// TIA Portal V19 export
VAR_GLOBAL   // PLC tag table "A02_201"
   A0201_Motore_Bancalata_1_Controllo_Connettore AT %I131.3 : Bool;   // 970X1A
   A0201_Banco_1_Phc_Ingresso AT %I131.4 : Bool;   // 973SQ1
   A0201_Banco_1_Phc_Uscita AT %I131.5 : Bool;   // 973SQ2
   "A0201_AUX_Spalla_1.1_Ls_Minimo" AT %I131.6 : Bool;   // 982SQ1
   "A0201_AUX_Spalla_1.1_Ls_Massimo" AT %I131.7 : Bool;   // 982SQ2
   "A0201_AUX_Spalla_1.2_Ls_Minimo" AT %I132.0 : Bool;   // 992SQ1
   "A0201_AUX_Spalla_1.2_Ls_Massimo" AT %I132.1 : Bool;   // 992SQ2
   "A0201_AUX_Spalla_1.3_Ls_Minimo" AT %I132.2 : Bool;   // 1002SQ1
   "A0201_AUX_Spalla_1.3_Ls_Massimo" AT %I132.3 : Bool;   // 1002SQ2
   "A0201_AUX_Spalla_1.4_Ls_Minimo" AT %I132.4 : Bool;   // 1006SQ1
   "A0201_AUX_Spalla_1.4_Ls_Massimo" AT %I132.5 : Bool;   // 1006SQ2
   A0201_Motore_Bancalata_2_Controllo_Connettore AT %I132.6 : Bool;   // 1020X1A
   A0201_Banco_2_Phc_Ingresso AT %I132.7 : Bool;   // 1023SQ1
   A0201_Banco_2_Phc_Uscita AT %I133.0 : Bool;   // 1023SQ2
   "A0201_AUX_Spalla_2.1_Ls_Minimo" AT %I133.1 : Bool;   // 1032SQ1
   "A0201_AUX_Spalla_2.1_Ls_Massimo" AT %I133.2 : Bool;   // 1032SQ2
   "A0201_AUX_Spalla_2.2_Ls_Minimo" AT %I133.3 : Bool;   // 1042SQ1
   "A0201_AUX_Spalla_2.2_Ls_Massimo" AT %I133.4 : Bool;   // 1042SQ2
   A0201_Motore_Bancalata_3_Lato_1_Controllo_Connettore AT %I133.5 : Bool;   // 1060X1A
   A0201_Banco_3_Lato_1_Phc_Ingresso AT %I133.6 : Bool;   // 1063SQ1
   A0201_Banco_3_Lato_1_Phc_Uscita AT %I133.7 : Bool;   // 1063SQ2
   "A0201_AUX_Spalla_3.1_Ls_Minimo_Apertura" AT %I134.0 : Bool;   // 1072SQ1
   "A0201_AUX_Spalla_3.1_Ls_Massimo_Apertura" AT %I134.1 : Bool;   // 1072SQ2
   "A0201_Spalla_3.3_Apre" AT %Q4.4 : Bool;   // 1080KM1
   "A0201_Spalla_3.3_Chiude" AT %Q4.5 : Bool;   // 1080KM2
   "A0201_Spalla_3.3_Anomalia_Termico" AT %I4.1 : Bool;   // 1080QF1
   "A0201_AUX_Spalla_3.3_Ls_Minimo_Apertura" AT %I134.2 : Bool;   // 1081SQ1
   "A0201_AUX_Spalla_3.3_Ls_Massimo_Apertura" AT %I134.3 : Bool;   // 1081SQ2
   "A0201_Spalla_3.5_Apre" AT %Q4.6 : Bool;   // 1085KM1
   "A0201_Spalla_3.5_Chiude" AT %Q4.7 : Bool;   // 1085KM2
   "A0201_Spalla_3.5_Anomalia_Termico" AT %I4.2 : Bool;   // 1085QF1
   "A0201_AUX_Spalla_3.5_Ls_Minimo_Apertura" AT %I134.4 : Bool;   // 1086SQ1
   "A0201_AUX_Spalla_3.5_Ls_Massimo_Apertura" AT %I134.5 : Bool;   // 1086SQ2
   "A0201_Spalla_3.7_Apre" AT %Q5.0 : Bool;   // 1090KM1
   "A0201_Spalla_3.7_Chiude" AT %Q5.1 : Bool;   // 1090KM2
   "A0201_AUX_Spalla_3.7_Ls_Minimo_Apertura" AT %I134.6 : Bool;   // 1091SQ1
   "A0201_AUX_Spalla_3.7_Ls_Massimo_Apertura" AT %I134.7 : Bool;   // 1091SQ2
   A0201_Motore_Bancalata_3_Lato_2_Controllo_Connettore AT %I135.0 : Bool;   // 1110X1A
   A0201_Banco_3_Lato_2_Phc_Ingresso AT %I135.1 : Bool;   // 1113SQ1
   A0201_Banco_3_Lato_2_Phc_Uscita AT %I135.2 : Bool;   // 1113SQ2
   "A0201_AUX_Spalla_3.2_Ls_Minimo" AT %I135.3 : Bool;   // 1122SQ1
   "A0201_AUX_Spalla_3.2_Ls_Massimo" AT %I135.4 : Bool;   // 1122SQ2
   "A0201_Spalla_3.4_Apre" AT %Q5.2 : Bool;   // 1130KM1
   "A0201_Spalla_3.4_Chiude" AT %Q5.3 : Bool;   // 1130KM2
   "A0201_Spalla_3.4_Anomalia_Termico" AT %I4.4 : Bool;   // 1130QF1
   "A0201_AUX_Spalla_3.4_Ls_Minimo" AT %I135.5 : Bool;   // 1131SQ1
   "A0201_AUX_Spalla_3.4_Ls_Massimo" AT %I135.6 : Bool;   // 1131SQ2
   "A0201_Spalla_3.6_Apre" AT %Q5.4 : Bool;   // 1135KM1
   "A0201_Spalla_3.6_Chiude" AT %Q5.5 : Bool;   // 1135KM2
   "A0201_Spalla_3.6_Anomalia_Termico" AT %I4.5 : Bool;   // 1135QF1
   "A0201_AUX_Spalla_3.6_Ls_Minimo" AT %I135.7 : Bool;   // 1136SQ1
   "A0201_AUX_Spalla_3.6_Ls_Massimo" AT %I136.0 : Bool;   // 1136SQ2
   "A0201_Spalla_3.8_Apre" AT %Q5.6 : Bool;   // 1140KM1
   "A0201_Spalla_3.8_Chiude" AT %Q5.7 : Bool;   // 1140KM2
   "A0201_Spalla_3.8_Anomalia_Termico" AT %I4.6 : Bool;   // 1140QF1
   "A0201_AUX_Spalla_3.8_Ls_Minimo" AT %I136.1 : Bool;   // 1141SQ1
   "A0201_AUX_Spalla_3.8_Ls_Massimo" AT %I136.2 : Bool;   // 1141SQ2
   A0201_Ventilatore_Mot_Profila_Marcia AT %Q1.5 : Bool;   // 1192QF1
   A0201_Ventilatore_Mot_Profila_Feedback AT %I4.7 : Bool;   // 1192KM1
   A0201_Phc_Inizio_Indroduttore_Profila AT %I136.3 : Bool;   // 1198SQ1
   A0201_Profila_Controllo_Bancale_Bit0 AT %I136.4 : Bool;   // 1204X1
   A0201_Profila_Controllo_Bancale_Bit1 AT %I136.5 : Bool;   // 1204X1
   A0201_Profila_Controllo_Bancale_Bit2 AT %I136.6 : Bool;   // 1204X1
   A0201_Profila_Phc_Prima_Encoder AT %I136.7 : Bool;   // 1204SQ1
   A0201_Profila_Phc_Dopo_Encoder AT %I137.0 : Bool;   // 1204SQ2
   A0201_Profila_Cassette_Pompa_Lubrificante_Marcia AT %Q1.6 : Bool;   // 1210QF1
   A0201_Profila_Cassette_Pompa_Lubrificante_Feedback AT %I5.0 : Bool;   // 1210KM1
   A0201_Profila_Cassette_V_Sezionatrice_Generale AT %Q140.0 : Bool;   // 1212YV1
   A0201_Profila_Cassette_Livello_Lubrificante AT %I137.1 : Bool;   // 1212SL1
   A0201_Profila_Cassetta_1_V_Lubrificante_1 AT %Q140.1 : Bool;   // 1214YV1
   A0201_Profila_Cassetta_1_V_Lubrificante_2 AT %Q140.2 : Bool;   // 1214YV2
   A0201_Profila_Cassetta_1_V_Lubrificante_3 AT %Q140.3 : Bool;   // 1214YV3
   A0201_Profila_Cassetta_1_V_Feedback_Lubrificante_1 AT %I137.2 : Bool;   // 1214SQ1
   A0201_Profila_Cassetta_1_V_Feedback_Lubrificante_2 AT %I137.3 : Bool;   // 1214SQ2
   A0201_Profila_Cassetta_1_V_Feedback_Lubrificante_3 AT %I137.4 : Bool;   // 1214SQ3
   A0201_Profila_Cassetta_1_V_Lubrificante_4 AT %Q140.4 : Bool;   // 1215YV1
   A0201_Profila_Cassetta_1_V_Lubrificante_5 AT %Q140.5 : Bool;   // 1215YV2
   A0201_Profila_Cassetta_1_V_Lubrificante_6 AT %Q140.6 : Bool;   // 1215YV3
   A0201_Profila_Cassetta_1_V_Feedback_Lubrificante_4 AT %I137.5 : Bool;   // 1215SQ1
   A0201_Profila_Cassetta_1_V_Feedback_Lubrificante_5 AT %I137.6 : Bool;   // 1215SQ2
   A0201_Profila_Cassetta_1_V_Feedback_Lubrificante_6 AT %I137.7 : Bool;   // 1215SQ3
   A0201_Profila_Cassetta_2_V_Lubrificante_1 AT %Q140.7 : Bool;   // 1218YV1
   A0201_Profila_Cassetta_2_V_Lubrificante_2 AT %Q141.0 : Bool;   // 1218YV2
   A0201_Profila_Cassetta_2_V_Lubrificante_3 AT %Q141.1 : Bool;   // 1218YV3
   A0201_Profila_Cassetta_2_V_Feedback_Lubrificante_1 AT %I138.0 : Bool;   // 1218SQ1
   A0201_Profila_Cassetta_2_V_Feedback_Lubrificante_2 AT %I138.1 : Bool;   // 1218SQ2
   A0201_Profila_Cassetta_2_V_Feedback_Lubrificante_3 AT %I138.2 : Bool;   // 1218SQ3
   A0201_Profila_Cassetta_2_V_Lubrificante_4 AT %Q141.2 : Bool;   // 1219YV1
   A0201_Profila_Cassetta_2_V_Lubrificante_5 AT %Q141.3 : Bool;   // 1219YV2
   A0201_Profila_Cassetta_2_V_Lubrificante_6 AT %Q141.4 : Bool;   // 1219YV3
   A0201_Profila_Cassetta_2_V_Feedback_Lubrificante_4 AT %I138.3 : Bool;   // 1219SQ1
   A0201_Profila_Cassetta_2_V_Feedback_Lubrificante_5_Libero AT %I138.4 : Bool;   // 1219SQ2
   A0201_Profila_Cassetta_2_V_Feedback_Lubrificante_6_Libero AT %I138.5 : Bool;   // 1219SQ3
   A0201_Profila_Cassetta_3_V_Lubrificante_1 AT %Q141.5 : Bool;   // 1222YV1
   A0201_Profila_Cassetta_3_V_Lubrificante_2 AT %Q141.6 : Bool;   // 1222YV2
   A0201_Profila_Cassetta_3_V_Lubrificante_3 AT %Q141.7 : Bool;   // 1222YV3
   A0201_Profila_Cassetta_3_V_Feedback_Lubrificante_1 AT %I138.6 : Bool;   // 1222SQ1
   A0201_Profila_Cassetta_3_V_Feedback_Lubrificante_2 AT %I138.7 : Bool;   // 1222SQ2
   A0201_Profila_Cassetta_3_V_Feedback_Lubrificante_3 AT %I139.0 : Bool;   // 1222SQ3
   A0201_Profila_Cassetta_3_V_Lubrificante_4 AT %Q142.0 : Bool;   // 1223YV1
   A0201_Profila_Cassetta_3_V_Lubrificante_5 AT %Q142.1 : Bool;   // 1223YV2
   A0201_Profila_Cassetta_3_V_Lubrificante_6 AT %Q142.2 : Bool;   // 1223YV3
   A0201_Profila_Cassetta_3_V_Feedback_Lubrificante_4 AT %I139.1 : Bool;   // 1223SQ1
   A0201_Profila_Cassetta_3_V_Feedback_Lubrificante_5_Libero AT %I139.2 : Bool;   // 1223SQ2
   A0201_Profila_Cassetta_3_V_Feedback_Lubrificante_6_Libero AT %I139.3 : Bool;   // 1223SQ3
   A0201_Fine_Profila_V_Soffio AT %Q142.3 : Bool;   // 1234YV1
   A0201_Fine_Profila_V_Soffio_Pulizia_Phc_Tacca AT %Q142.4 : Bool;   // 1234YV2
   A0201_Ls_Controllo_Inceppamento AT %I139.4 : Bool;   // 1243SQ1
   A0201_Carrello_Riposizionatore_Phc_Prima_Encoder AT %I139.5 : Bool;   // 1245SQ1
   A0201_Carrello_Misuratore_Posizione_Zero AT %I139.6 : Bool;   // 1245SQ2
   A0201_Carrello_Misuratore_Rallentamento_Verso_Zero AT %I139.7 : Bool;   // 1245SQ3
   A0201_Carrello_Misuratore_Rallentamento_Verso_Posizione_Rest AT %I140.0 : Bool;   // 1245SQ4
   A0201_Carrello_Misuratore_Stop_Verso_Rest AT %I140.1 : Bool;   // 1245SQ5
   A0201_Carrello_Misuratore_Posizione_Work AT %I140.2 : Bool;   // 1245SQ6
   A0201_Carrello_Misuratore_In_Appoggio_Tra_Loro AT %I140.3 : Bool;   // 1245SQ7
   A0201_Carrello_Riposizionatore_Phc_Dopo_Encoder AT %I140.4 : Bool;   // 1245SQ8
   A0201_Pinza_Misuratore_V_Rest AT %Q104.1 : Bool;   // 1246YV1
   A0201_Pinza_Misuratore_V_Work AT %Q104.2 : Bool;   // 1246YV2
   A0201_Pinza_Misuratore_Ls_Rest AT %I140.5 : Bool;   // 1246SQ1
   A0201_Pinza_Misuratore_Ls_Work AT %I140.6 : Bool;   // 1246SQ2
   "A0201_Taglio_Al_Volo_V_Lubrificazione_Chioccola+Pattini" AT %Q142.5 : Bool;   // 1306YV1
   A0201_Taglio_Al_Volo_Livello_Lubririficazione AT %I140.7 : Bool;   // 1306SL1
   A0201_Centralina_Olio_Banco_Taglio_Anomalie_Termici AT %I5.1 : Bool;   // 1320FR1
   A0201_AUX_Centralina_Olio_Banco_Taglio_Potenza AT %Q1.7 : Bool;   // 1322KA1
   A0201_AUX_Centralina_Olio_Banco_Taglio_Conferma_Triangolo AT %I5.2 : Bool;   // 1320KM3
   A0201_AUX_Centralina_Olio_Banco_Taglio_Minimo_Minimo_Allarme_Grave AT %I141.0 : Bool;   // 1326SL1
   A0201_AUX_Centralina_Olio_Banco_Taglio_Minimo_Allarme_Lieve AT %I141.1 : Bool;   // 1326SL2
   "A0201_AUX_Centralina_Olio_Banco_Taglio_Max_Temperatura_70°C" AT %I141.2 : Bool;   // 1326S1
   A0201_Ricircolo_Centralina_Olio_Banco_Taglio_Marcia AT %Q2.0 : Bool;   // 1328QF1
   A0201_Ricircolo_Centralina_Olio_Banco_Taglio_Feedback AT %I5.3 : Bool;   // 1328KM1
   A0201_Ricircolo_Centralina_Olio_Banco_Taglio_Filtro_Intasato AT %I141.3 : Bool;   // 1328S1
   A0201_Ventilatore_Centralina_Olio_Banco_Taglio_Marcia AT %Q2.1 : Bool;   // 1330QF1
   A0201_Ventilatore_Centralina_Olio_Banco_Taglio_Feedback AT %I5.4 : Bool;   // 1330KM1
   A0201_V_Bloccaggio_Matrici_Testa_Taglio_T1_Rest AT %Q104.3 : Bool;   // 1350YV1
   A0201_V_Bloccaggio_Matrici_Testa_Taglio_T1_Work AT %Q104.4 : Bool;   // 1350YV2
   A0201_Testa_Taglio_T1_V_Rest AT %Q104.5 : Bool;   // 1351YV1
   A0201_Testa_Taglio_T1_V_Work AT %Q104.6 : Bool;   // 1351YV2
   A0201_Testa_Taglio_T1_Ls_Rest AT %I141.4 : Bool;   // 1351SQ1
   A0201_Testa_Taglio_T1_Ls_Work AT %I141.5 : Bool;   // 1351SQ2
   A0201_Testa_Imbottitura_T2_V_Rest AT %Q104.7 : Bool;   // 1352YV1
   A0201_Testa_Imbottitura_T2_V_Work AT %Q105.0 : Bool;   // 1352YV2
   A0201_Testa_Imbottitura_T2_Ls_Rest AT %I141.6 : Bool;   // 1352SQ1
   A0201_Testa_Imbottitura_T2_Ls_Work AT %I141.7 : Bool;   // 1352SQ2
   A0201_Testa_Marchiatura_T3_V_Rest AT %Q105.1 : Bool;   // 1353YV1
   A0201_Testa_Marchiatura_T3_V_Work AT %Q105.2 : Bool;   // 1353YV2
   A0201_Testa_Marchiatura_T3_Ls_Rest AT %I142.0 : Bool;   // 1353SQ1
   A0201_Testa_Marchiatura_T3_Ls_Work AT %I142.1 : Bool;   // 1353SQ2
   A0201_Testa_Libero_T4_V_Rest AT %Q105.3 : Bool;   // 1354YV1
   A0201_Testa_Libero_T4_V_Work AT %Q105.4 : Bool;   // 1354YV2
   A0201_Testa_Libero_T4_Ls_Rest AT %I142.2 : Bool;   // 1354
   A0201_Testa_Libero_T4_Ls_Work AT %I142.3 : Bool;   // 1354
   A0201_Stampi_Fine_Linea_V_Lubrificazione AT %Q142.6 : Bool;   // 1360YV1
   A0201_Stampi_Fine_Linea_Livello_Lubrificante AT %I142.4 : Bool;   // 1360SL1
   A0201_Centralina_Olio_Banco_Taglio_AI_Pressione AT %IW916 : Int;
   A0201_Centralina_Olio_Banco_Taglio_AI_Temperatura AT %IW918 : Int;
   A0201_Banco_Taglio_AI_Pressione_Testa_T1 AT %IW920 : Int;
   "Area02_Anomalie_Termico_Spalla_1.3" AT %I3.7 : Bool;   // 1000QF1
   "A0201_Spalla_1.4_Anomalia_Termico" AT %I4.0 : Bool;   // 1005QF1
   "A0201_Spalla_3.7_Anomalia_Termico" AT %I4.3 : Bool;   // 1090QF1
   "A0201_Spalla_1.3_Apre" AT %Q4.0 : Bool;   // 1000KM1
   "A0201_Spalla_1.3_Chiude" AT %Q4.1 : Bool;   // 1000KM1
   "A0201_Spalla_1.4_Apre" AT %Q4.2 : Bool;
   "A0201_Spalla_1.4_Chiude" AT %Q4.3 : Bool;
END_VAR
